FUNCTION_BLOCK FB_UpdateHandler
VAR_INPUT
	I_SekUpdate			:BOOL;
	I_SekReset			:BOOL;
	I_SysUpdate			:BOOL;
	I_SysReset			:BOOL;
END_VAR

VAR_OUTPUT
	O_SekUpdate			:BOOL;
	O_SysUpdate			:BOOL;
END_VAR
VAR 
	SekSwitch			:SR;
	SysSwitch			:SR;
END_VAR

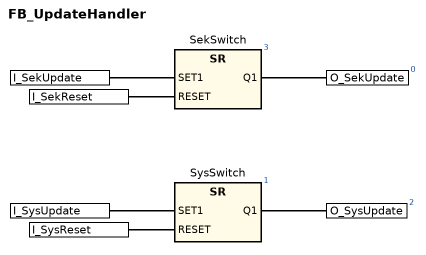
O_SekUpdate := SekSwitch.Q1;
SysSwitch(SET1 := I_SysUpdate, RESET := I_SysReset); // SR
O_SysUpdate := SysSwitch.Q1;
SekSwitch(SET1 := I_SekUpdate, RESET := I_SekReset); // SR

END_FUNCTION_BLOCK

(* stored: Version 1.1.0.1, ProductVersion 3.1.4024.12
   POU FB_UpdateHandler: Id {9b0f81e2-b778-4353-8739-91d96e1c742a}, SpecialFunc None *)
